// TIA Portal V15.1 export
// export: Created 2024-06-21T08:41:24.9669167Z, ExportSetting WithDefaults, DisplayName Totally Integrated Automation Portal, DisplayVersion V15.1 Update 5, DisplayName TIA Portal Openness, DisplayVersion V15.1 Update 5, DisplayName SINAMICS Startdrive Advanced, DisplayVersion V15.1, DisplayName G130, G150, S120, S150, SINAMICS MV, S210, DisplayVersion V15.1, DisplayName G110M, G120, G120C, G120D, G120P, DisplayVersion V15.1, DisplayName STEP 7 Professional, DisplayVersion V15.1 Update 5, DisplayName STEP 7 Safety, DisplayVersion V15.1, DisplayName WinCC Professional, DisplayVersion V15.1 Update 5, DisplayName SIMATIC Visualization Architect, DisplayVersion V15.1
FUNCTION "209230ZM01Orders" : Void   // FC403, FBD
TITLE = 209230ZM01Orders
{ S7_Optimized_Access := 'FALSE' }
AUTHOR : VCC
VERSION : 0.1
// stored: AutoNumber false, IsIECCheckEnabled false, SetENOAutomatically False, UDAEnableTagReadback false
   VAR_OUTPUT
      O_AlarmA : Bool;   // Alarm A
      O_AlarmB : Bool;   // Alarm B
      O_AlarmC : Bool;   // Alarm C
      O_AlarmD : Bool;   // Alarm D
      O_AlarmABCondition : Bool;   // Alarm AB Condition
      H_IAnim : DWord;   // Icon Animation
   END_VAR
   VAR_TEMP
      TempDint : DInt;
   END_VAR
   VAR_TEMP   // added for the SCL form of the ladder/FBD networks
      _w1 : Bool;
   END_VAR
BEGIN

REGION Network 1: **** 4.6 - Machine Status - Indication **** Icon Animation
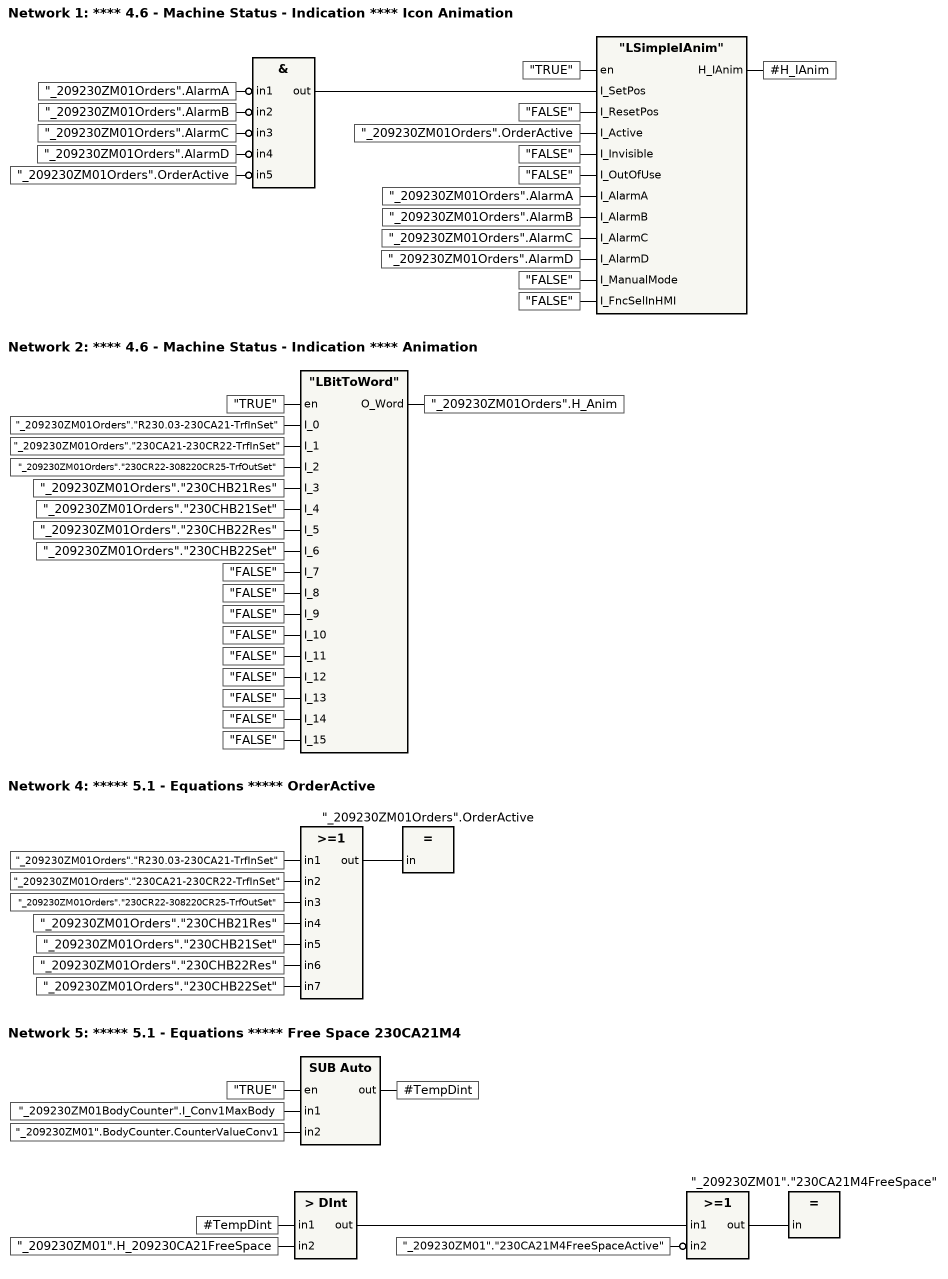
   IF "TRUE" THEN
       "LSimpleIAnim"(I_SetPos := NOT "_209230ZM01Orders".AlarmA AND NOT "_209230ZM01Orders".AlarmB AND NOT "_209230ZM01Orders".AlarmC AND NOT "_209230ZM01Orders".AlarmD AND NOT "_209230ZM01Orders".OrderActive,
                      I_ResetPos := "FALSE",
                      I_Active := "_209230ZM01Orders".OrderActive,
                      I_Invisible := "FALSE",
                      I_OutOfUse := "FALSE",
                      I_AlarmA := "_209230ZM01Orders".AlarmA,
                      I_AlarmB := "_209230ZM01Orders".AlarmB,
                      I_AlarmC := "_209230ZM01Orders".AlarmC,
                      I_AlarmD := "_209230ZM01Orders".AlarmD,
                      I_ManualMode := "FALSE",
                      I_FncSelInHMI := "FALSE",
                      H_IAnim => #H_IAnim);
   END_IF;
END_REGION

REGION Network 2: **** 4.6 - Machine Status - Indication **** Animation
   IF "TRUE" THEN
       "LBitToWord"(I_0 := "_209230ZM01Orders"."R230.03-230CA21-TrfInSet",
                    I_1 := "_209230ZM01Orders"."230CA21-230CR22-TrfInSet",
                    I_2 := "_209230ZM01Orders"."230CR22-308220CR25-TrfOutSet",
                    I_3 := "_209230ZM01Orders"."230CHB21Res",
                    I_4 := "_209230ZM01Orders"."230CHB21Set",
                    I_5 := "_209230ZM01Orders"."230CHB22Res",
                    I_6 := "_209230ZM01Orders"."230CHB22Set",
                    I_7 := "FALSE",
                    I_8 := "FALSE",
                    I_9 := "FALSE",
                    I_10 := "FALSE",
                    I_11 := "FALSE",
                    I_12 := "FALSE",
                    I_13 := "FALSE",
                    I_14 := "FALSE",
                    I_15 := "FALSE",
                    O_Word => "_209230ZM01Orders".H_Anim);
   END_IF;
END_REGION

NETWORK
TITLE = **** 4.6 - Machine Status - Indications **** Animation DB number
// DB number
      OPN   "_209230ZM01Orders";
      L     DBNO;
      T     "_209230ZM01Orders".H_DBnr;

REGION Network 4: ***** 5.1 - Equations ***** OrderActive
   "_209230ZM01Orders".OrderActive := "_209230ZM01Orders"."R230.03-230CA21-TrfInSet" OR "_209230ZM01Orders"."230CA21-230CR22-TrfInSet" OR "_209230ZM01Orders"."230CR22-308220CR25-TrfOutSet" OR "_209230ZM01Orders"."230CHB21Res" OR "_209230ZM01Orders"."230CHB21Set" OR "_209230ZM01Orders"."230CHB22Res" OR "_209230ZM01Orders"."230CHB22Set";
END_REGION

REGION Network 5: ***** 5.1 - Equations ***** Free Space 230CA21M4
   IF "TRUE" THEN
       #TempDint := "_209230ZM01BodyCounter".I_Conv1MaxBody - "_209230ZM01".BodyCounter.CounterValueConv1;
   END_IF;
   "_209230ZM01"."230CA21M4FreeSpace" := (#TempDint > "_209230ZM01".H_209230CA21FreeSpace) OR NOT "_209230ZM01"."230CA21M4FreeSpaceActive";
END_REGION

REGION Network 6: ***** 5.1 - Equations ***** Body between 220CA21M4SG2 and 220CA21M4SG4
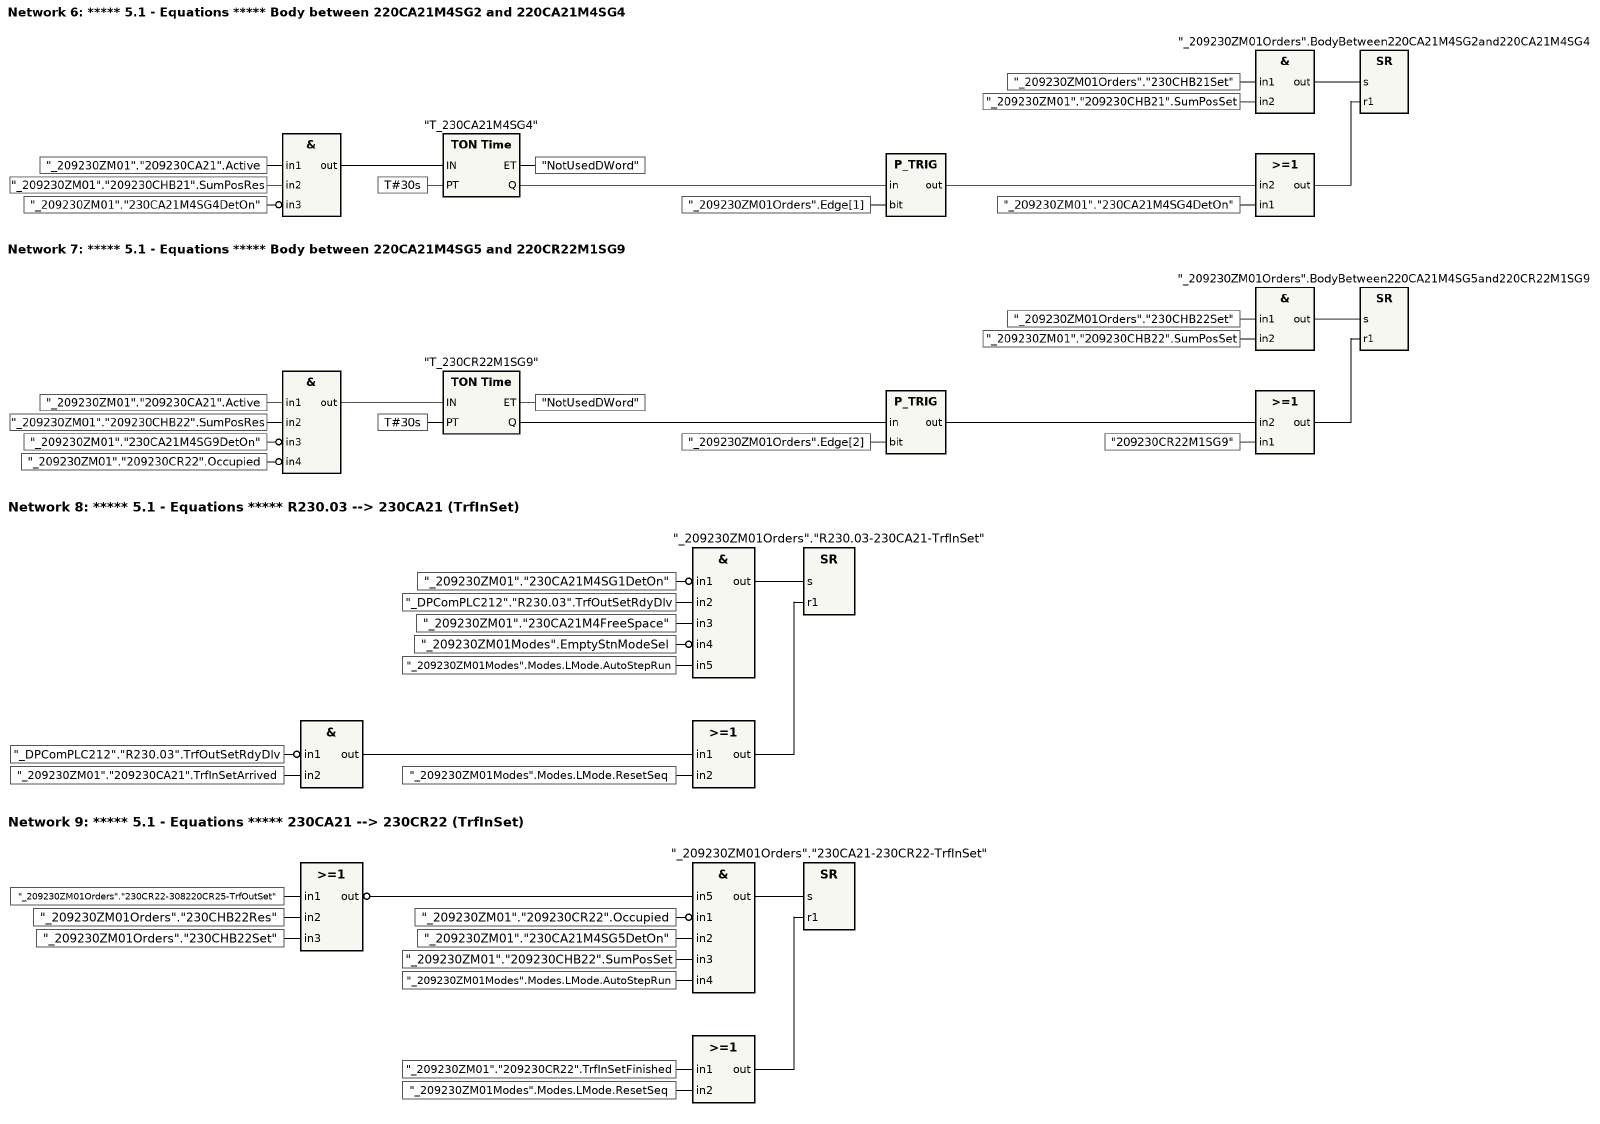
   "T_230CA21M4SG4".TON(IN := "_209230ZM01"."209230CA21".Active AND "_209230ZM01"."209230CHB21".SumPosRes AND NOT "_209230ZM01"."230CA21M4SG4DetOn",
                        PT := T#30s,
                        ET => "NotUsedDWord");
   #_w1 := "T_230CA21M4SG4".Q AND NOT "_209230ZM01Orders".Edge[1];   // rising edge
   "_209230ZM01Orders".Edge[1] := "T_230CA21M4SG4".Q;
   IF "_209230ZM01Orders"."230CHB21Set" AND "_209230ZM01"."209230CHB21".SumPosSet THEN
       "_209230ZM01Orders".BodyBetween220CA21M4SG2and220CA21M4SG4 := TRUE;   // SR flip-flop
   END_IF;
   IF #_w1 OR "_209230ZM01"."230CA21M4SG4DetOn" THEN
       "_209230ZM01Orders".BodyBetween220CA21M4SG2and220CA21M4SG4 := FALSE;
   END_IF;
END_REGION

REGION Network 7: ***** 5.1 - Equations ***** Body between 220CA21M4SG5 and 220CR22M1SG9
   "T_230CR22M1SG9".TON(IN := "_209230ZM01"."209230CA21".Active AND "_209230ZM01"."209230CHB22".SumPosRes AND NOT "_209230ZM01"."230CA21M4SG9DetOn" AND NOT "_209230ZM01"."209230CR22".Occupied,
                        PT := T#30s,
                        ET => "NotUsedDWord");
   #_w1 := "T_230CR22M1SG9".Q AND NOT "_209230ZM01Orders".Edge[2];   // rising edge
   "_209230ZM01Orders".Edge[2] := "T_230CR22M1SG9".Q;
   IF "_209230ZM01Orders"."230CHB22Set" AND "_209230ZM01"."209230CHB22".SumPosSet THEN
       "_209230ZM01Orders".BodyBetween220CA21M4SG5and220CR22M1SG9 := TRUE;   // SR flip-flop
   END_IF;
   IF #_w1 OR "209230CR22M1SG9" THEN
       "_209230ZM01Orders".BodyBetween220CA21M4SG5and220CR22M1SG9 := FALSE;
   END_IF;
END_REGION

REGION Network 8: ***** 5.1 - Equations ***** R230.03 --> 230CA21 (TrfInSet)
   IF NOT "_209230ZM01"."230CA21M4SG1DetOn" AND "_DPComPLC212"."R230.03".TrfOutSetRdyDlv AND "_209230ZM01"."230CA21M4FreeSpace" AND NOT "_209230ZM01Modes".EmptyStnModeSel AND "_209230ZM01Modes".Modes.LMode.AutoStepRun THEN
       "_209230ZM01Orders"."R230.03-230CA21-TrfInSet" := TRUE;   // SR flip-flop
   END_IF;
   IF (NOT "_DPComPLC212"."R230.03".TrfOutSetRdyDlv AND "_209230ZM01"."209230CA21".TrfInSetArrived) OR "_209230ZM01Modes".Modes.LMode.ResetSeq THEN
       "_209230ZM01Orders"."R230.03-230CA21-TrfInSet" := FALSE;
   END_IF;
END_REGION

REGION Network 9: ***** 5.1 - Equations ***** 230CA21 --> 230CR22 (TrfInSet)
   IF NOT ("_209230ZM01Orders"."230CR22-308220CR25-TrfOutSet" OR "_209230ZM01Orders"."230CHB22Res" OR "_209230ZM01Orders"."230CHB22Set") AND NOT "_209230ZM01"."209230CR22".Occupied AND "_209230ZM01"."230CA21M4SG5DetOn" AND "_209230ZM01"."209230CHB22".SumPosSet AND "_209230ZM01Modes".Modes.LMode.AutoStepRun THEN
       "_209230ZM01Orders"."230CA21-230CR22-TrfInSet" := TRUE;   // SR flip-flop
   END_IF;
   IF "_209230ZM01"."209230CR22".TrfInSetFinished OR "_209230ZM01Modes".Modes.LMode.ResetSeq THEN
       "_209230ZM01Orders"."230CA21-230CR22-TrfInSet" := FALSE;
   END_IF;
END_REGION

REGION Network 10: ***** 5.1 - Equations ***** 230CR22 --> 308220CR25 (TrfOutSet)
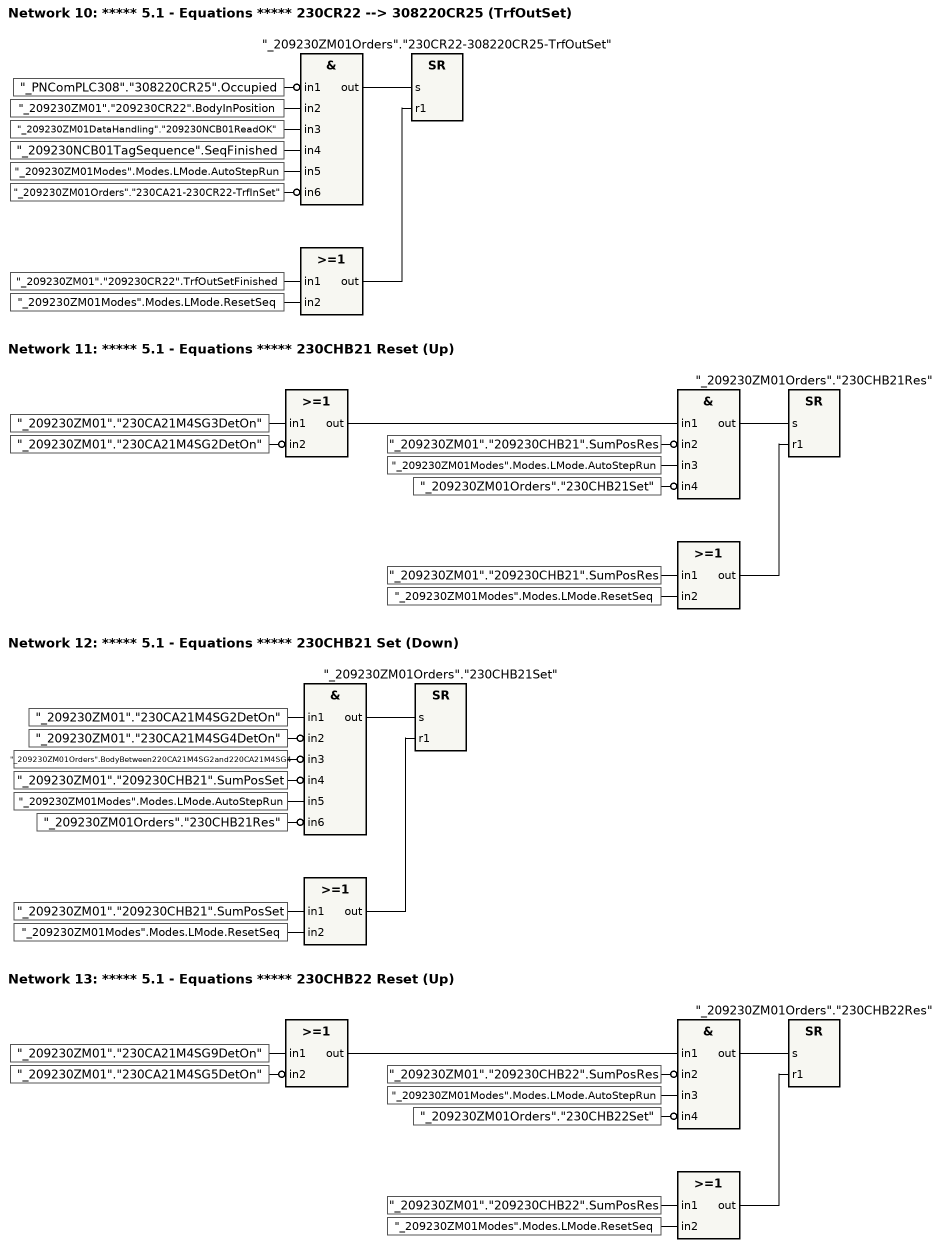
   IF NOT "_PNComPLC308"."308220CR25".Occupied AND "_209230ZM01"."209230CR22".BodyInPosition AND "_209230ZM01DataHandling"."209230NCB01ReadOK" AND "_209230NCB01TagSequence".SeqFinished AND "_209230ZM01Modes".Modes.LMode.AutoStepRun AND NOT "_209230ZM01Orders"."230CA21-230CR22-TrfInSet" THEN
       "_209230ZM01Orders"."230CR22-308220CR25-TrfOutSet" := TRUE;   // SR flip-flop
   END_IF;
   IF "_209230ZM01"."209230CR22".TrfOutSetFinished OR "_209230ZM01Modes".Modes.LMode.ResetSeq THEN
       "_209230ZM01Orders"."230CR22-308220CR25-TrfOutSet" := FALSE;
   END_IF;
END_REGION

REGION Network 11: ***** 5.1 - Equations ***** 230CHB21 Reset (Up)
   IF ("_209230ZM01"."230CA21M4SG3DetOn" OR NOT "_209230ZM01"."230CA21M4SG2DetOn") AND NOT "_209230ZM01"."209230CHB21".SumPosRes AND "_209230ZM01Modes".Modes.LMode.AutoStepRun AND NOT "_209230ZM01Orders"."230CHB21Set" THEN
       "_209230ZM01Orders"."230CHB21Res" := TRUE;   // SR flip-flop
   END_IF;
   IF "_209230ZM01"."209230CHB21".SumPosRes OR "_209230ZM01Modes".Modes.LMode.ResetSeq THEN
       "_209230ZM01Orders"."230CHB21Res" := FALSE;
   END_IF;
END_REGION

REGION Network 12: ***** 5.1 - Equations ***** 230CHB21 Set (Down)
   IF "_209230ZM01"."230CA21M4SG2DetOn" AND NOT "_209230ZM01"."230CA21M4SG4DetOn" AND NOT "_209230ZM01Orders".BodyBetween220CA21M4SG2and220CA21M4SG4 AND NOT "_209230ZM01"."209230CHB21".SumPosSet AND "_209230ZM01Modes".Modes.LMode.AutoStepRun AND NOT "_209230ZM01Orders"."230CHB21Res" THEN
       "_209230ZM01Orders"."230CHB21Set" := TRUE;   // SR flip-flop
   END_IF;
   IF "_209230ZM01"."209230CHB21".SumPosSet OR "_209230ZM01Modes".Modes.LMode.ResetSeq THEN
       "_209230ZM01Orders"."230CHB21Set" := FALSE;
   END_IF;
END_REGION

REGION Network 13: ***** 5.1 - Equations ***** 230CHB22 Reset (Up)
   IF ("_209230ZM01"."230CA21M4SG9DetOn" OR NOT "_209230ZM01"."230CA21M4SG5DetOn") AND NOT "_209230ZM01"."209230CHB22".SumPosRes AND "_209230ZM01Modes".Modes.LMode.AutoStepRun AND NOT "_209230ZM01Orders"."230CHB22Set" THEN
       "_209230ZM01Orders"."230CHB22Res" := TRUE;   // SR flip-flop
   END_IF;
   IF "_209230ZM01"."209230CHB22".SumPosRes OR "_209230ZM01Modes".Modes.LMode.ResetSeq THEN
       "_209230ZM01Orders"."230CHB22Res" := FALSE;
   END_IF;
END_REGION

REGION Network 14: ***** 5.1 - Equations ***** 230CHB22 Set (Down)
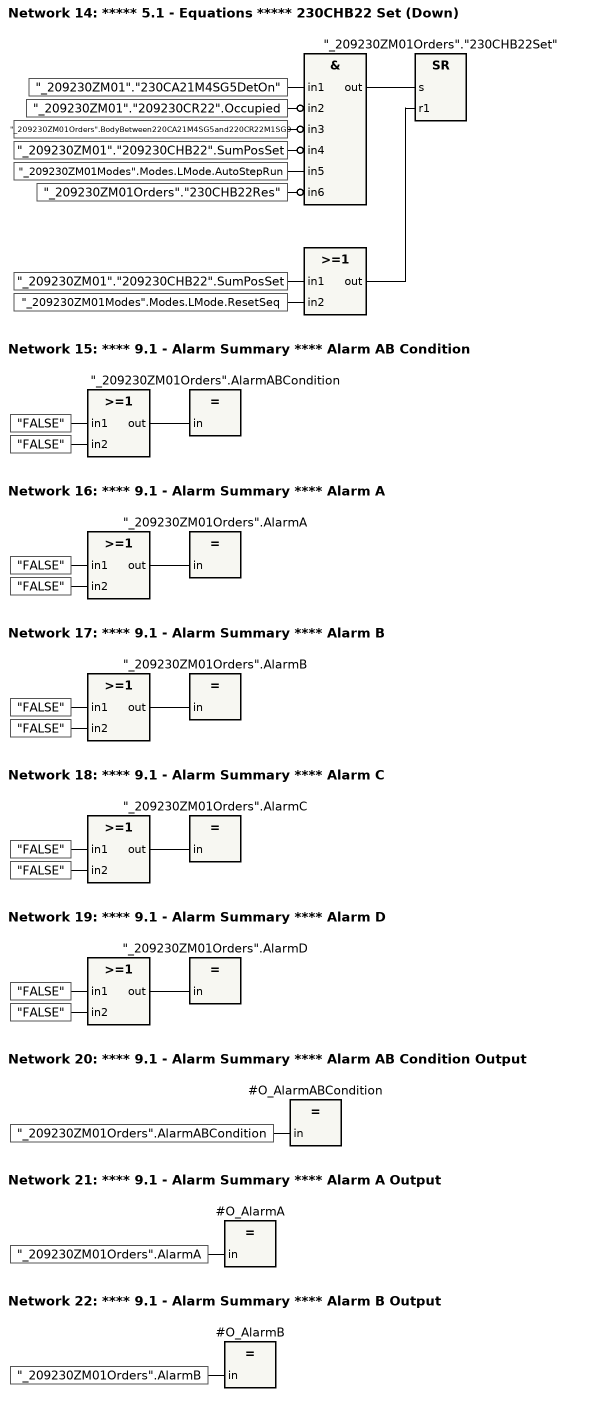
   IF "_209230ZM01"."230CA21M4SG5DetOn" AND NOT "_209230ZM01"."209230CR22".Occupied AND NOT "_209230ZM01Orders".BodyBetween220CA21M4SG5and220CR22M1SG9 AND NOT "_209230ZM01"."209230CHB22".SumPosSet AND "_209230ZM01Modes".Modes.LMode.AutoStepRun AND NOT "_209230ZM01Orders"."230CHB22Res" THEN
       "_209230ZM01Orders"."230CHB22Set" := TRUE;   // SR flip-flop
   END_IF;
   IF "_209230ZM01"."209230CHB22".SumPosSet OR "_209230ZM01Modes".Modes.LMode.ResetSeq THEN
       "_209230ZM01Orders"."230CHB22Set" := FALSE;
   END_IF;
END_REGION

REGION Network 15: **** 9.1 - Alarm Summary **** Alarm AB Condition
   "_209230ZM01Orders".AlarmABCondition := "FALSE" OR "FALSE";
END_REGION

REGION Network 16: **** 9.1 - Alarm Summary **** Alarm A
   "_209230ZM01Orders".AlarmA := "FALSE" OR "FALSE";
END_REGION

REGION Network 17: **** 9.1 - Alarm Summary **** Alarm B
   "_209230ZM01Orders".AlarmB := "FALSE" OR "FALSE";
END_REGION

REGION Network 18: **** 9.1 - Alarm Summary **** Alarm C
   "_209230ZM01Orders".AlarmC := "FALSE" OR "FALSE";
END_REGION

REGION Network 19: **** 9.1 - Alarm Summary **** Alarm D
   "_209230ZM01Orders".AlarmD := "FALSE" OR "FALSE";
END_REGION

REGION Network 20: **** 9.1 - Alarm Summary **** Alarm AB Condition Output
   #O_AlarmABCondition := "_209230ZM01Orders".AlarmABCondition;
END_REGION

REGION Network 21: **** 9.1 - Alarm Summary **** Alarm A Output
   #O_AlarmA := "_209230ZM01Orders".AlarmA;
END_REGION

REGION Network 22: **** 9.1 - Alarm Summary **** Alarm B Output
   #O_AlarmB := "_209230ZM01Orders".AlarmB;
END_REGION

REGION Network 23: **** 9.1 - Alarm Summary **** Alarm C Output
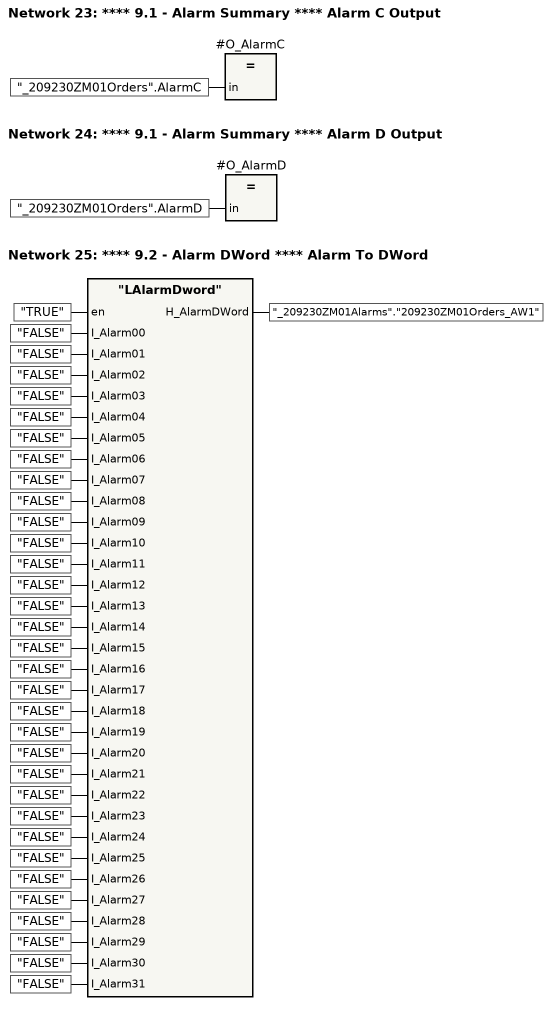
   #O_AlarmC := "_209230ZM01Orders".AlarmC;
END_REGION

REGION Network 24: **** 9.1 - Alarm Summary **** Alarm D Output
   #O_AlarmD := "_209230ZM01Orders".AlarmD;
END_REGION

REGION Network 25: **** 9.2 - Alarm DWord **** Alarm To DWord
   // Alarm Word
   IF "TRUE" THEN
       "LAlarmDword"(I_Alarm00 := "FALSE",
                     I_Alarm01 := "FALSE",
                     I_Alarm02 := "FALSE",
                     I_Alarm03 := "FALSE",
                     I_Alarm04 := "FALSE",
                     I_Alarm05 := "FALSE",
                     I_Alarm06 := "FALSE",
                     I_Alarm07 := "FALSE",
                     I_Alarm08 := "FALSE",
                     I_Alarm09 := "FALSE",
                     I_Alarm10 := "FALSE",
                     I_Alarm11 := "FALSE",
                     I_Alarm12 := "FALSE",
                     I_Alarm13 := "FALSE",
                     I_Alarm14 := "FALSE",
                     I_Alarm15 := "FALSE",
                     I_Alarm16 := "FALSE",
                     I_Alarm17 := "FALSE",
                     I_Alarm18 := "FALSE",
                     I_Alarm19 := "FALSE",
                     I_Alarm20 := "FALSE",
                     I_Alarm21 := "FALSE",
                     I_Alarm22 := "FALSE",
                     I_Alarm23 := "FALSE",
                     I_Alarm24 := "FALSE",
                     I_Alarm25 := "FALSE",
                     I_Alarm26 := "FALSE",
                     I_Alarm27 := "FALSE",
                     I_Alarm28 := "FALSE",
                     I_Alarm29 := "FALSE",
                     I_Alarm30 := "FALSE",
                     I_Alarm31 := "FALSE",
                     H_AlarmDWord => "_209230ZM01Alarms"."209230ZM01Orders_AW1");
   END_IF;
END_REGION
END_FUNCTION
